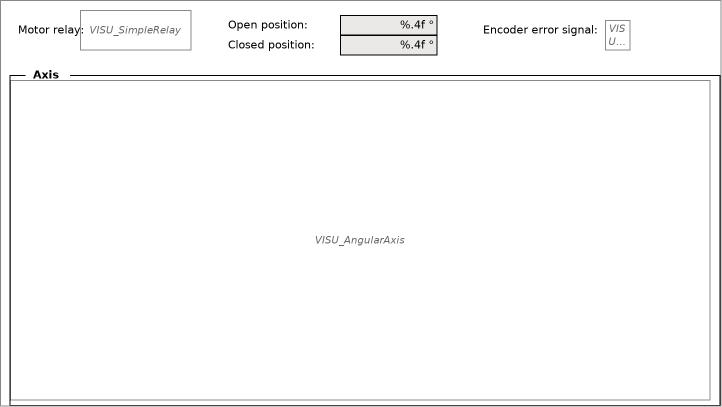
VISUALIZATION VISU_CoverPanel  // 722x407
VAR_IN_OUT
    panelConfig : CoverPanelConfig;
	panel : CoverPanel;
    widget : CoverPanelWidget;
END_VAR
    Label (225,15 90x20), "Open position:"
    Rectangle (340,15 97x20), "%.4f °", text variable: panelConfig.openPosition
    Label (225,35 90x20), "Closed position:"
    Rectangle (340,35 97x20), "%.4f °", text variable: panelConfig.closedPosition
    Frame (80,10 111x40)
        shows VISU_SimpleRelay(ref := panel.parts.motorRelay, widget := widget.motorRelay)
    Label (15,15 95x30), "Motor relay:"
    Frame (10,80 700x320)
        shows VISU_AngularAxis(axis := panel.parts.axis, widget := widget.axis)
    Line (10,75) (25,75)
    Label (30,65 45x20), "Axis"
    Line (70,75) (720,75)
    Line (720,405) (720,75)
    Line (10,405) (720,405)
    Line (10,405) (10,75)
    Label (480,15 130x30), "Encoder error signal:"
    Frame (605,20 25x30)
        shows VISU_State_gray_red(state := panel.encoderErrorSignal)
END_VISUALIZATION

(* stored: Version 1.1.0.1, ProductVersion 3.1.4019.2
   Visu VISU_CoverPanel: Id {f38b25c3-b51d-4ac9-9193-db45209a13bd} *)
